FUNCTION_BLOCK AnalogueTerminal IMPLEMENTS ITF_Analogue
VAR
	_SomeValueFromIO : INT := 8192;
END_VAR

METHOD GetValue : LREAL
VAR_INPUT
END_VAR
GetValue :=  (_SomeValueFromIO/32767.0)*10.0;
END_METHOD

END_FUNCTION_BLOCK

(* stored: Version 1.1.0.1, ProductVersion 3.1.4024.12
   POU AnalogueTerminal: Id {4488c845-3d30-4fbe-b94d-3166a97201e0}, SpecialFunc None
   Method GetValue: Id {d33fb718-9046-4669-824b-90df2621771c} *)
